FUNCTION TryConvert_LREAL_TO_SINT : BOOL
VAR_INPUT
	in : LREAL;
	out : REFERENCE TO SINT;
END_VAR

IF in > DatatypeLimits.MAX_VALUE_OF_LREAL_WHICH_CAN_BE_HELD_IN_A_SINT THEN
	RETURN;
END_IF

IF in < DatatypeLimits.MIN_VALUE_OF_LREAL_WHICH_CAN_BE_HELD_IN_A_SINT THEN
	RETURN;
END_IF

out := LREAL_TO_SINT(in);
TryConvert_LREAL_TO_SINT := TRUE;

END_FUNCTION

(* stored: Version 1.1.0.1, ProductVersion 3.1.4024.12
   POU TryConvert_LREAL_TO_SINT: Id {cadc5d7d-f2f9-4937-8deb-da6f13f6678c}, SpecialFunc None *)
